// TIA Portal V16 export
// export: Created 2022-09-05T21:51:21.6557122Z, ExportSetting WithDefaults, DisplayName Totally Integrated Automation Portal, DisplayVersion V16, DisplayName TIA Portal Version Control Interface, DisplayVersion V16, DisplayName TIA Portal Openness, DisplayVersion V16, DisplayName SINAMICS Startdrive Advanced, DisplayVersion V16, DisplayName SINAMICS Startdrive G130, G150, S120, S150, SINAMICS MV, S210, DisplayVersion V16, DisplayName SINAMICS Startdrive G110M, G120, G120C, G120D, G120P, DisplayVersion V16, DisplayName STEP 7 Professional, DisplayVersion V16, DisplayName STEP 7 Safety, DisplayVersion V16, DisplayName WinCC Professional, DisplayVersion V16
VAR_GLOBAL   // PLC tag table "Counter_Table"
   stop AT %I0.0 : Bool;
   start AT %I0.1 : Bool;
   system AT %M0.0 : Bool;
   box_conveyor AT %Q0.0 : Bool;
   box_sensor AT %I0.2 : Bool;
   apple_conveyor AT %Q0.1 : Bool;
   apple_sensor AT %I0.3 : Bool;
END_VAR
